PROGRAM P_Adapter
VAR
	cylinderStandard				: Cylinder;
	cylinderVtem					: CylinderVtem;
END_VAR


// Move cylinders forward
cylinderStandard.fwd();
cylinderVtem.fwd();

END_PROGRAM

(* stored: Version 1.1.0.1, ProductVersion 3.1.4024.12
   POU P_Adapter: Id {40cba971-86e8-4d4c-8cef-ebe86ac679f0}, SpecialFunc None *)
